TYPE JsonDoc : STRING( JsonParams.JSON_DOC_SIZE ); END_TYPE

(* stored: Version 1.1.0.1, ProductVersion 3.1.4022.18
   DUT JsonDoc: Id {d9f2df7f-705f-00eb-2bc4-bfeb90739c39} *)
